(* LS Electric XG5000 project: XMC_MultiAxis_FBs *)
(* sample programs for multi-axis function blocks. *)
(* PLC LSPLC *)
(* module base 0 slot 0: Input/Output Module:XMC-DN24 (DC 24V Input 8Points/TR output 16Points) *)
(* module base 0 slot 1: Internal Analog Input/Output:XMF-AH04E (A/D voltage/current 2 channels, D/A voltage 2 channels) *)
(* task Periodic Task: Kind=2 *)
(* task Initialization Task: Kind=1 *)
(* task NC Program: Kind=6 *)

PROGRAM ECAT_Connect_Example (* task: Scan Program *)
(* example of LS_Connect and LS_Disconnect function blocks *)
VAR
    Execute_Connect : BOOL; (* Execute LS_Connect function block *)
    Execute_Disconnect : BOOL; (* Execute LS_Disconnect *)
    INST_LS_CONNECT : LS_CONNECT; (* Instance of LS_Connect function block *)
    INST_LS_DISCONNECT : LS_DISCONNECT; (* LS_Disconnect function block instance *)
END_VAR
(* AutomationDirect.com has provided this code for convenience. This sample code is provided "as-is" with no expressed or implied warranty. 
 If the end user includes any of the sample code (in whole or part), it is the user's responsibility to completely modify, integrate, and test any code to ensure it meets all system and 
 safety requirements for the intended application or system. *)

//Example of LS_Connect Function block to connect EtherCAT network
INST_LS_CONNECT(Execute:=Execute_Connect, ErrorID=>INST_LS_CONNECT.ErrorID);

//Example of LS_Disconnect Function block to disconnect the EtherCAT network
INST_LS_DISCONNECT(Execute:=Execute_Disconnect, ErrorID=>INST_LS_DISCONNECT.ErrorID);
END_PROGRAM

PROGRAM MC_PowerAll_Example (* task: Scan Program *)
(* ST Example of MC_PowerAll function block *)
VAR
    All_Axes_Ready : BOOL; (* Status that all axes are ready *)
    INST_MC_POWERALL : MC_POWERALL; (* Instance of MC_PowerAll function block *)
    Power_On_Axes : BOOL; (* command to power on all axes *)
END_VAR
//Check that all axes are ready
IF (_AX01_SV_RDY) AND (_AX02_SV_RDY) AND (_AX03_SV_RDY) AND (_AX04_SV_RDY) THEN
	All_Axes_Ready := TRUE;
ELSE
	All_Axes_Ready := FALSE;
END_IF;

//check that it is good to run MC_PowerAll
IF (All_Axes_Ready) THEN
	//Example of MC_PowerAll function block
	INST_MC_POWERALL(Enable:=Power_On_Axes, ErrorID=>INST_MC_POWERALL.ErrorID);
END_IF;
END_PROGRAM

PROGRAM Home_Example (* task: Scan Program *)
(* ST example for MC_HomeAll and LS_HomeAll function blocks *)
VAR
    All_Axes_Pwr_On : BOOL; (* All axes are powered on *)
    All_Axes_Ready : BOOL; (* All axes are ready *)
    Execute_LSHomeAll : BOOL; (* Execute LS_HomeAll function block *)
    Execute_MCHomeAll : BOOL; (* execute MC_HomeAll function block *)
    Home_Position : LREAL; (* position of axex after homing *)
    Homing_Method : SINT; (* Homing Method for LS_HomeAll *)
    INST_LS_HOMEALL : LS_HOMEALL; (* LS_HomeAll function block instance *)
    INST_MC_HOMEALL : MC_HOMEALL; (* instance of MC_HomeAll function block *)
END_VAR
//Check that all axes are ready
IF (_AX01_RDY) AND (_AX02_RDY) AND (_AX03_RDY) AND (_AX04_RDY) THEN
	All_Axes_Ready := TRUE;
ELSE
	All_Axes_Ready := FALSE;
END_IF;

//Check that all axes are powered on
IF (_AX01_SV_ON) AND (_AX02_SV_ON) AND (_AX03_SV_ON) AND (_AX04_SV_ON) THEN
	All_Axes_Pwr_On := TRUE;
ELSE
	All_Axes_Pwr_On := FALSE;
END_IF;

//Make sure axes are ready
IF (All_Axes_Pwr_On) AND (All_Axes_Ready) THEN
	
	//Example of MC_HomeAll function block
	INST_MC_HOMEALL(Execute:=Execute_MCHomeAll, Position:=Home_Position, BufferMode:=0, ErrorID=>INST_MC_HOMEALL.ErrorID);
	
	
	//Example of LS_HomeAll function block
	INST_LS_HOMEALL(Execute:=Execute_LSHomeAll, Position:=Home_Position, HomingMethod:=Homing_Method, SwitchSearchSpeed:=1000.0, 
		ZeroSearchSpeed:=100.0, HomingAcc:=100.0, HomeOffset:=0.0, DoneBehavior:=0, BufferMode:=0, ErrorID=>INST_LS_HOMEALL.ErrorID);
END_IF;
END_PROGRAM

PROGRAM MCStopAll_MCHaltAll_Example (* task: Scan Program *)
(* Example of MC_StopAll and MC_HaltAll function blocks *)
VAR
    All_Axes_Pwr_On : BOOL; (* All axes are powered on *)
    All_Axes_Ready : BOOL; (* All axes are ready *)
    Execute_HaltAll : BOOL; (* Execute MC_HaltAll function block *)
    Execute_StopAll : BOOL; (* execute MC_StopAll function block *)
    INST_MC_HALTALL : MC_HALTALL; (* instance of MC_HaltAll function block *)
    INST_MC_STOPALL : MC_STOPALL; (* Instance of MC_StopAll function block *)
END_VAR
//Check that all axes are ready
IF (_AX01_RDY) AND (_AX02_RDY) AND (_AX03_RDY) AND (_AX04_RDY) THEN
	All_Axes_Ready := TRUE;
ELSE
	All_Axes_Ready := FALSE;
END_IF;

//Check that all axes are powered on
IF (_AX01_SV_ON) AND (_AX02_SV_ON) AND (_AX03_SV_ON) AND (_AX04_SV_ON) THEN
	All_Axes_Pwr_On := TRUE;
ELSE
	All_Axes_Pwr_On := FALSE;
END_IF;


IF (All_Axes_Pwr_On) AND (All_Axes_Ready) THEN
	//Example of MC_StopAll function block
	INST_MC_STOPALL(Execute:=Execute_StopAll, Deceleration:=10000.0, Jerk:=1000.0, ErrorID=>INST_MC_STOPALL.ErrorID);
	
	//Example of MC_HaltAll function block
	INST_MC_HALTALL(Execute:=Execute_HaltAll, Deceleration:=10000.0, Jerk:=1000.0, BufferMode:=0, ErrorID=>INST_MC_HALTALL.ErrorID);
END_IF;
END_PROGRAM

PROGRAM MC_Reset2All_Example2 (* task: Scan Program *)
(* ST example of MC_Reset2All function block *)
VAR
    All_Axes_Ready : BOOL; (* status that all axes are ready *)
    Execute_ResetAll : BOOL; (* execute the MC_Reset2All function block *)
    INST_MC_RESET2ALL : MC_RESET2ALL; (* MC_Reset2All function block instance *)
END_VAR
//Check that all axes are ready
IF (_AX01_SV_RDY) AND (_AX02_SV_RDY) AND (_AX03_SV_RDY) AND (_AX04_SV_RDY) THEN
	All_Axes_Ready := TRUE;
ELSE
	All_Axes_Ready := FALSE;
END_IF;

IF (All_Axes_Ready) THEN
	//Example of MC_Reset2All function block
	INST_MC_RESET2ALL(Execute:=Execute_ResetAll, ErrorType:=2, ErrorID=>INST_MC_RESET2ALL.ErrorID);
END_IF;
END_PROGRAM

PROGRAM MC_CamIn_CamOut_Example (* task: Scan Program *)
(* ST version of MC_CamIn and MC_CamOut function blocks *)
VAR
    All_Axes_Pwr_On : BOOL; (* all axes are powered on *)
    All_Axes_Ready : BOOL; (* all axes are ready *)
    Execute_CamIn : BOOL; (* execute the MC_CamIn fb *)
    Execute_CamOut : BOOL; (* execute MC_CamOut function block *)
    Execute_MasterMove : BOOL; (* execute master move velocity *)
    Master_Axis : UINT; (* Master axis for camming *)
    Master_MOVEVELOCITY : MC_MOVEVELOCITY; (* fb for master move velocity command *)
    Slave_Axis : UINT; (* slave axis for camming *)
    Slave_CAMIN : MC_CAMIN; (* fb instance for slave camin *)
    Slave_CAMOUT : MC_CAMOUT; (* MC_CamOut for slave axis *)
END_VAR
//Check that all axes are ready
IF (_AX01_RDY) AND (_AX02_RDY)  THEN
	All_Axes_Ready := TRUE;
ELSE
	All_Axes_Ready := FALSE;
END_IF;

//Check that all axes are powered on
IF (_AX01_SV_ON) AND (_AX02_SV_ON)  THEN
	All_Axes_Pwr_On := TRUE;
ELSE
	All_Axes_Pwr_On := FALSE;
END_IF;

//Set MasterAxis and SlaveAxis variables
Master_Axis := 2;
Slave_Axis := 1;

IF (All_Axes_Pwr_On) AND (All_Axes_Ready) THEN
	//MoveVelocity command for master axis
	Master_MOVEVELOCITY(Execute:=Execute_MasterMove, Axis:=Master_Axis, ContinuousUpdate:=0, Velocity:=50000.0, Acceleration:=10000.0, 
		Deceleration:=10000.0, Jerk:=1000.0, Direction:=1, BufferMode:=0, ErrorID=>Master_MOVEVELOCITY.ErrorID);
	
	//MC_CamIn for Slave axis
	Slave_CAMIN(Execute:=Execute_CamIn, Master:=Master_Axis, Slave:=Slave_Axis, ContinuousUpdate:=0, MasterOffset:=Slave_CAMIN.MasterOffset, 
		SlaveOffset:=Slave_CAMIN.SlaveOffset, MasterScaling:=Slave_CAMIN.MasterScaling, SlaveScaling:=Slave_CAMIN.SlaveScaling, 
		MasterStartDistance:=Slave_CAMIN.MasterStartDistance, MasterSyncPosition:=Slave_CAMIN.MasterSyncPosition, StartMode:=Slave_CAMIN.StartMode, 
		MasterValueSource:=Slave_CAMIN.MasterValueSource, CamTableID:=Slave_CAMIN.CamTableID, BufferMode:=0, ErrorID=>Slave_CAMIN.ErrorID);
	
	
	//MC_CamOut example - disengage the camming of the slave
	Slave_CAMOUT(Execute:=Execute_CamOut, Slave:=Slave_Axis, ErrorID=>Slave_CAMOUT.ErrorID);
END_IF;
END_PROGRAM

PROGRAM MC_GearIn_GearInEx_GearOut (* task: Scan Program *)
(* ST example of MC_GearIn, MC_GearInEx, and MC_GearOut *)
VAR
    All_Axes_Pwr_On : BOOL; (* all axes are powered on *)
    All_Axes_Ready : BOOL; (* all axes are ready *)
    Execute_GearIn : BOOL; (* execute MC_GearIn fb *)
    Execute_GearInEx : BOOL; (* execute MC_GearInEx fb *)
    Execute_GearOut : BOOL; (* execute MC_GearOut fb *)
    Execute_MasterMove : BOOL; (* execute master MC_MoveVelocity *)
    Master_Axis : UINT; (* master axis for gear in *)
    Master_MOVEVELOCITY : MC_MOVEVELOCITY; (* master MC_MoveVelocity fb *)
    Slave_Axis : UINT; (* slave axis for gear in *)
    Slave_GEARIN : MC_GEARIN; (* MC_GearIn for Slave axis *)
    Slave_GEARINEX : MC_GEARINEX; (* MC_GearInEx for slave axis *)
    Slave_GEAROUT : MC_GEAROUT; (* MC_GearOut for slave axis *)
END_VAR
//Check that all axes are ready
IF (_AX01_RDY) AND (_AX02_RDY)  THEN
	All_Axes_Ready := TRUE;
ELSE
	All_Axes_Ready := FALSE;
END_IF;

//Check that all axes are powered on
IF (_AX01_SV_ON) AND (_AX02_SV_ON)  THEN
	All_Axes_Pwr_On := TRUE;
ELSE
	All_Axes_Pwr_On := FALSE;
END_IF;

//Set MasterAxis and SlaveAxis variables
Master_Axis := 2;
Slave_Axis := 1;


IF (All_Axes_Pwr_On) AND (All_Axes_Ready) THEN
	
	//MoveVelocity command for master axis
	Master_MOVEVELOCITY(Execute:=Execute_MasterMove, Axis:=Master_Axis, ContinuousUpdate:=0, Velocity:=50000.0, Acceleration:=10000.0, 
		Deceleration:=10000.0, Jerk:=1000.0, Direction:=1, BufferMode:=0, ErrorID=>Master_MOVEVELOCITY.ErrorID);
	
	//Example MC_GearIn fb
	Slave_GEARIN(Execute:=Execute_GearIn, Master:=Master_Axis, Slave:=Slave_Axis, ContinuousUpdate:=0, RatioNumerator:=Slave_GEARIN.RatioNumerator, 
		RatioDenominator:=Slave_GEARIN.RatioDenominator, MasterValueSource:=Slave_GEARIN.MasterValueSource, Acceleration:=Slave_GEARIN.Acceleration, 
		Deceleration:=Slave_GEARIN.Deceleration, Jerk:=Slave_GEARIN.Jerk, BufferMode:=0, ErrorID=>Slave_GEARIN.ErrorID);
	
	//Example MC_GearInEx fb
	Slave_GEARINEX(Execute:=Execute_GearInEx, Master:=Master_Axis, Slave:=Slave_Axis, ContinuousUpdate:=0, RatioNumerator:=Slave_GEARINEX.RatioNumerator, 
		RatioDenominator:=Slave_GEARINEX.RatioDenominator, MasterValueSource:=Slave_GEARINEX.MasterValueSource, Acceleration:=Slave_GEARINEX.Acceleration, 
		Deceleration:=Slave_GEARINEX.Deceleration, Jerk:=Slave_GEARINEX.Jerk, BufferMode:=0, ErrorID=>Slave_GEARINEX.ErrorID);
	
	//Example MC_GearOut fb
	Slave_GEAROUT(Execute:=Execute_GearOut, Slave:=Slave_Axis, ErrorID=>Slave_GEAROUT.ErrorID);
END_IF;
END_PROGRAM

PROGRAM MC_GearInPos_GearInPosEx (* task: Scan Program *)
(* ST example of MC_GearInPos and MC_GearInPosEx *)
VAR
    All_Axes_Pwr_On : BOOL; (* all axes are powered on *)
    All_Axes_Ready : BOOL; (* all axes are ready *)
    Execute_GearInPos : BOOL; (* execute MC_GearInPos *)
    Execute_GearInPosEx : BOOL; (* execute MC_GearInPosEx fb *)
    Execute_MoveRelative : BOOL; (* execute master MC_MoveAbsolute *)
    Master_Axis : UINT; (* master axis *)
    Master_MOVERELATIVE : MC_MOVERELATIVE; (* master MC_MoveRelative *)
    Slave_Axis : UINT; (* slave axis *)
    Slave_GEARINPOS : MC_GEARINPOS; (* slave axis MC_GearInPos *)
    Slave_GEARINPOSEX : MC_GEARINPOSEX; (* MC_GearInPosEx for slave axis *)
END_VAR
//Check that all axes are ready
IF (_AX01_RDY) AND (_AX02_RDY)  THEN
	All_Axes_Ready := TRUE;
ELSE
	All_Axes_Ready := FALSE;
END_IF;

//Check that all axes are powered on
IF (_AX01_SV_ON) AND (_AX02_SV_ON)  THEN
	All_Axes_Pwr_On := TRUE;
ELSE
	All_Axes_Pwr_On := FALSE;
END_IF;

//Set MasterAxis and SlaveAxis variables
Master_Axis := 2;
Slave_Axis := 1;

IF (All_Axes_Pwr_On) AND (All_Axes_Ready) THEN
	//Move Absolute for master
	Master_MOVERELATIVE(Execute:=Execute_MoveRelative, Axis:=Master_Axis, ContinuousUpdate:=0, Distance:=2000000.0, Velocity:=50000.0, Acceleration:=50000.0, 
		Deceleration:=50000.0, Jerk:=1000.0, BufferMode:=0, ErrorID=>Master_MOVERELATIVE.ErrorID);
	
	//MC_GearInPos fb example
	Slave_GEARINPOS(Execute:=Execute_GearInPos, Master:=Master_Axis, Slave:=Slave_Axis, RatioNumerator:=Slave_GEARINPOS.RatioNumerator, 
		RatioDenominator:=Slave_GEARINPOS.RatioDenominator, MasterValueSource:=Slave_GEARINPOS.MasterValueSource, MasterSyncPosition:=Slave_GEARINPOS.MasterSyncPosition, 
		SlaveSyncPosition:=Slave_GEARINPOS.SlaveSyncPosition, SyncMode:=0, MasterStartDistance:=Slave_GEARINPOS.MasterStartDistance, Velocity:=Slave_GEARINPOS.Velocity, 
		Acceleration:=Slave_GEARINPOS.Acceleration, Deceleration:=Slave_GEARINPOS.Deceleration, Jerk:=Slave_GEARINPOS.Jerk, BufferMode:=0, ErrorID=>Slave_GEARINPOS.ErrorID);
	
	//MC_GearInPosEx fb example
	Slave_GEARINPOSEX(Execute:=Execute_GearInPosEx, Master:=Master_Axis, Slave:=Slave_Axis, RatioNumerator:=Slave_GEARINPOSEX.RatioNumerator, 
		RatioDenominator:=Slave_GEARINPOSEX.RatioDenominator, MasterValueSource:=Slave_GEARINPOSEX.MasterValueSource, MasterSyncPosition:=Slave_GEARINPOSEX.MasterSyncPosition, 
		SlaveSyncPosition:=Slave_GEARINPOSEX.SlaveSyncPosition, SyncMode:=0, MasterStartDistance:=Slave_GEARINPOSEX.MasterStartDistance, Velocity:=Slave_GEARINPOSEX.Velocity, 
		Acceleration:=Slave_GEARINPOSEX.Acceleration, Deceleration:=Slave_GEARINPOSEX.Deceleration, Jerk:=Slave_GEARINPOSEX.Jerk, BufferMode:=0, ErrorID=>Slave_GEARINPOSEX.ErrorID);
END_IF;
END_PROGRAM

PROGRAM MC_Phasing_Example (* task: Scan Program *)
(* ST Example of MC_Phasing *)
VAR
    All_Axes_Pwr_On : BOOL; (* all axes are powered on *)
    All_Axes_Ready : BOOL; (* status that all axes are ready *)
    Execute_Phasing : BOOL; (* execute MC_Phasing fb *)
    Master_Axis : UINT; (* Master axis *)
    Slave_Axis : UINT; (* slave axis *)
    Slave_PHASING : MC_PHASING; (* MC_Phasing function block instance *)
END_VAR
//Check that all axes are ready
IF (_AX01_RDY) AND (_AX02_RDY)  THEN
	All_Axes_Ready := TRUE;
ELSE
	All_Axes_Ready := FALSE;
END_IF;

//Check that all axes are powered on
IF (_AX01_SV_ON) AND (_AX02_SV_ON)  THEN
	All_Axes_Pwr_On := TRUE;
ELSE
	All_Axes_Pwr_On := FALSE;
END_IF;

//Set MasterAxis and SlaveAxis variables
Master_Axis := 2;
Slave_Axis := 1;


IF (All_Axes_Pwr_On) AND (All_Axes_Ready) THEN
	//Example of MC_Phasing fb
	Slave_PHASING(Execute:=Execute_Phasing, Master:=Master_Axis, Slave:=Slave_Axis, PhaseShift:=Slave_PHASING.PhaseShift, Velocity:=Slave_PHASING.Velocity, 
		Acceleration:=Slave_PHASING.Acceleration, Deceleration:=Slave_PHASING.Deceleration, Jerk:=Slave_PHASING.Jerk, ErrorID=>Slave_PHASING.ErrorID);
END_IF;
END_PROGRAM

PROGRAM MC_SetPositionAll_Example2 (* task: Scan Program *)
(* ST example for MC_SetPositionAll *)
VAR
    All_Axes_Ready : BOOL; (* all axes are ready *)
    Execute_SetPosition : BOOL; (* Execute MC_SetPositionAll fb *)
    INST_MC_SETPOSITIONALL : MC_SETPOSITIONALL; (* MC_SetPositionAll fb *)
END_VAR
//Check that all axes are ready
IF (_AX01_RDY) AND (_AX02_RDY) AND (_AX03_RDY) AND (_AX04_RDY) THEN
	All_Axes_Ready := TRUE;
ELSE
	All_Axes_Ready := FALSE;
END_IF;

IF (All_Axes_Ready) THEN
	//Example of MC_SetPositionAll
	INST_MC_SETPOSITIONALL(Execute:=Execute_SetPosition, Position:=INST_MC_SETPOSITIONALL.Position, Relative:=INST_MC_SETPOSITIONALL.Relative, 
		ExecutionMode:=INST_MC_SETPOSITIONALL.ExecutionMode, ErrorID=>INST_MC_SETPOSITIONALL.ErrorID);
END_IF;
END_PROGRAM